INTERFACE ITF_TopElement2_HMI EXTENDS ITF_BaseTopElement_HMI

END_INTERFACE

(* stored: Version 1.1.0.1, ProductVersion 3.1.4024.15
   Itf ITF_TopElement2_HMI: Id {a8f92e7b-2e87-460e-af5c-b6c890ab43ea} *)
